FUNCTION LPF_FilterInit
VAR_INPUT
	CutFreq : REAL;
	Filter : POINTER TO LowPassFilter;
	TS : REAL;
END_VAR
VAR
END_VAR

Filter^.FrequencyCut := CutFreq;
Filter^.CutFreq := 1/1/(2*3.1415*Filter^.FrequencyCut);


Filter^.Den := 1/(TS + 2*(Filter^.CutFreq));
	
Filter^.a1 := (TS - 2*Filter^.CutFreq)*Filter^.Den;
Filter^.b0 := TS*Filter^.Den;
Filter^.b1 := TS*Filter^.Den;

END_FUNCTION

(* stored: Version 1.1.0.1, ProductVersion 3.1.4024.4
   POU LPF_FilterInit: Id {1027333b-fc50-4dfb-bf6a-660cb3466cb2}, SpecialFunc None *)
